{attribute 'qualified_only'}
{attribute 'strict'}
{attribute 'to_string'}
TYPE E_Season :
(
    Autumn,
    Winter,
    Spring,
    Summer
);
END_TYPE

(* stored: Version 1.1.0.1, ProductVersion 3.1.4024.12
   DUT E_Season: Id {5c24e66a-4c5a-0ed6-2319-d63e7906765f} *)
